{attribute 'qualified_only'}
{attribute 'strict'}
TYPE eSchedulerMode :
(
	continous := 0,
	daily := 1,
	weekly := 2
);
END_TYPE

(* stored: Version 1.1.0.1, ProductVersion 3.1.4026.18
   DUT eSchedulerMode: Id {82faea09-d953-4eef-a719-7a1598cc0ed4} *)
